FUNCTION_BLOCK FB_Foerderband
VAR_INPUT
	bEnable : BOOL;
	bExecute : BOOL;
	bHalt : BOOL;
END_VAR

VAR_OUTPUT
	eState : eBetriebszustand;
END_VAR
VAR
	nState : INT := 0;
	rVelocity : REAL;
	rAcceleration : REAL;
	// Motionblöcke der Tc2_Mc2
	mcReset : MC_Reset;
	mcPower : MC_Power;
	mcVelocity : MC_MoveVelocity;
	mcHalt : MC_Halt;
END_VAR

VAR_IN_OUT
	ax : Axis_Ref;
END_VAR

ax.ReadStatus();
mcReset(
	Axis:= ax, 
	Execute:= , 
	Done=> , 
	Busy=> , 
	Error=> , 
	ErrorID=> );
	
mcPower(
	Axis:= ax, 
	Enable:= , 
	Enable_Positive:= , 
	Enable_Negative:= , 
	Override:= , 
	BufferMode:= , 
	Options:= , 
	Status=> , 
	Busy=> , 
	Error=> , 
	ErrorID=> );

mcVelocity(
	Axis:= ax, 
	Execute:= , 
	Velocity:= 30, 
	Acceleration:= 60, 
	Deceleration:= , 
	Jerk:= , 
	Direction:= MC_Positive_Direction, 
	BufferMode:= , 
	Options:= , 
	InVelocity=> , 
	Busy=> , 
	Active=> , 
	CommandAborted=> , 
	Error=> , 
	ErrorID=> );
	
mcHalt(
	Axis:= ax, 
	Execute:= , 
	Deceleration:= 60, 
	Jerk:= , 
	BufferMode:= , 
	Options:= , 
	Done=> , 
	Busy=> , 
	Active=> , 
	CommandAborted=> , 
	Error=> , 
	ErrorID=> );
	
IF NOT mcPower.Status THEN
	nState := 0;
END_IF

CASE nState OF
	
END_CASE

END_FUNCTION_BLOCK

(* stored: Version 1.1.0.1, ProductVersion 3.1.4024.15
   POU FB_Foerderband: Id {2819a62a-8874-4d2c-b723-f866df5fb0bc}, SpecialFunc None *)
